PROGRAM Controller_PRG
VAR
END_VAR

END_PROGRAM

(* stored: Version 1.1.0.1, ProductVersion 3.1.4022.7
   POU Controller_PRG: Id {d7ffc0b2-bea9-4071-b871-ad534ffebbe7}, SpecialFunc None *)
